FUNCTION_BLOCK Test_F_PadString_TruncsLongStrings EXTENDS T_UnitTestBase
VAR
    SubjectString : T_MaxString;
    ResultString  : T_MaxString;
END_VAR

METHOD Init
VAR_INPUT
END_VAR
END_METHOD

{attribute 'analysis' := '-33'} // inhibit unused variable warning
METHOD RunTest
SubjectString := 'A long message with too many characters';
ResultString  := F_PadString(InputString := SubjectString,
                             Length      := 20);

AssertEquals_INT(Expected := 20,
                 Actual   := LEN(ResultString),
                 Message  := 'LEN(ResultString)');

AssertEquals_STRING(Expected := 'A long message with ',
                    Actual   := ResultString,
                    Message  := 'ResultString');

TestCompleted := TRUE;
END_METHOD

END_FUNCTION_BLOCK

(* stored: Version 1.1.0.1, ProductVersion 3.1.4024.12
   POU Test_F_PadString_TruncsLongStrings: Id {277b310f-45dc-4306-844b-b4d7121604ac}, SpecialFunc None
   Method Init: Id {a44d22eb-9f4f-05dd-1d32-46f1ee5392d1}
   Method RunTest: Id {a5072636-c388-0fa5-24dd-0ac984e14ca8} *)
